Universal Robots PolyScope program: ATI Simple Demo Program.urp

Program ATI Simple Demo Program (createdIn=3.4.1.292 lastSavedIn=3.3.0.145 directory=/home/ur/ursim-3.3.0/programs installation=default robotSerialNumber=2014359999)
Calibrated DH parameters: a=[0.000241, -0.156882, -0.391168, -0.000034, 0.000033, 0]; d=[0.08909, 1210.353649, -1202.089359, -8.154207, 0.094912, 0.082482]; alpha=[1.570962, 0.000326, -0.003342, 1.570446, -1.570439, 0]; deltaTheta=[0.000082, 1.192638, -1.263181, 0.0705, 0.00007, 0.000052]
BeforeStart
  Folder Move to initial start position
    MoveJ speed 60 deg/s, acceleration 80 deg/s^2 (recalculateMotions=false)
      Waypoint Start: TCP in base x=-436.825 y=579.513 z=220.778 mm, rx=3.1381 ry=-0.1132 rz=-0.0056 rad; joints [-61.803, -57.175, 58.456, -91.289, 270.047, 29.954] deg; flange x=-436.348 y=579.679 z=355.315 mm, rx=3.1399 ry=-0.0472 rz=-0.0055 rad
    URCap com.ur.urcap.ATI_FT.ATI FT Sensor data=running = Enable
Robot Program (runOnlyOnce=false motionType=MoveJ speed=1.047198 acceleration=1.396263 recalculateMotions=false)
  Folder Bias the sensor
    Wait Sleep waitTime=1
    URCap com.ur.urcap.ATI_FT.ATI FT Sensor data=running = Bias
  MoveL speed 50 mm/s, acceleration 400 mm/s^2 (recalculateMotions=false) feature=Base
    Folder Move down until the tool touches a surface
      If force()<2 (checkContinuously=true)
        Waypoint End (Relative): relativeFromPosition TCP in base x=-436.852 y=579.502 z=220.847 mm, rx=3.1382 ry=-0.1131 rz=-0.0056 rad; joints [-61.803, -57.175, 58.456, -91.289, 270.047, 29.954] deg; TCP in base x=-436.822 y=579.49 z=91.266 mm, rx=3.1382 ry=-0.1129 rz=-0.0055 rad; joints [-61.791, -53.885, 72.402, -108.525, 270.053, 29.909] deg; flange x=-436.348 y=579.679 z=225.723 mm, rx=3.1399 ry=-0.0472 rz=-0.0055 rad
    Folder Wait, then return to the start position
      Wait Sleep waitTime=1
      Waypoint Start: TCP in base x=-436.825 y=579.513 z=220.778 mm, rx=3.1381 ry=-0.1132 rz=-0.0056 rad; joints [-61.803, -57.175, 58.456, -91.289, 270.047, 29.954] deg; flange x=-436.348 y=579.679 z=355.315 mm, rx=3.1399 ry=-0.0472 rz=-0.0055 rad
Thread Thread_1 (runOnlyOnce=false trackProgramExecution=false)
  ForceMagnitude := force()
  Wait Sleep waitTime=0.1
